PROGRAM MAIN
VAR CONSTANT
  Dofs : ARRAY [0..3] OF INT := [1, 3, 6, 7];
  IterationCount : INT := 5;
  TrajactoryCount : DINT := 64 * 1024;
END_VAR
VAR
  _positionDist : RandomGaussian(seed:=42, mu:=0, sigma:=4);
  _dynamicDist : RandomGaussian(seed:=43, mu:=0, sigma:=0.8);
  _limitDist : RandomUniform(seed:=44, lowerBound:=0, upperBound:=4);
  
  _p : Randomizer(_positionDist);
  _d : Randomizer(_dynamicDist);
  _l : Randomizer(_limitDist);
  
  _otg : Struckig.Ruckig(0.001);
  _input : Struckig.InputParameter(0);
  _output : Struckig.OutputParameter;
  
  _step : INT := 0;
  _dt, _it, _jt : DINT := 0;
  
  _trajectoryStatistic, _itStatistic, _worstStatistic : MovingStatistic;
  
  _averageMean, _worstMean, _averageSigma, _worstSigma : ARRAY[0..3] OF LREAL; 
  
  _cpucounter : Tc2_System.GETCPUACCOUNT;
END_VAR

REPEAT
  CASE _step
  OF
    // setup ****************************************************
    0: 
    // **********************************************************
      
      _input.FB_init(TRUE, TRUE, dofs:=Dofs[_dt]);
      _trajectoryStatistic.Reset();
      _itStatistic.Reset();
      _worstStatistic.Reset();
      
      _p.Fill(ADR(_input.CurrentPosition), Dofs[_dt]);
      _p.Fill(ADR(_input.TargetPosition), Dofs[_dt]);
      _l.FillMax(ADR(_input.maxVelocity), Dofs[_dt], ADR(_input.TargetVelocity));
      _l.FillMax(ADR(_input.maxAcceleration), Dofs[_dt], ADR(_input.TargetAcceleration));
      _l.Fill(ADR(_input.maxJerk), Dofs[_dt]);
      CheckCalculation(_otg, _input);  
    
      _step := 1;
  
    // iterate start ********************************************
    1: 
    // **********************************************************
    
      _trajectoryStatistic.Reset();
      _step := 2;
      
    // iterate loop *********************************************
    2: 
    // **********************************************************
    
      _p.Fill(ADR(_input.CurrentPosition), Dofs[_dt]);
      _d.FillOrZero(ADR(_input.CurrentVelocity), Dofs[_dt], 0.9);
      _d.FillOrZero(ADR(_input.CurrentAcceleration), Dofs[_dt], 0.8);
      _p.Fill(ADR(_input.TargetPosition), Dofs[_dt]);
      _d.FillOrZero(ADR(_input.TargetVelocity), Dofs[_dt], 0.7);
      _d.FillOrZero(ADR(_input.TargetAcceleration), Dofs[_dt], 0.6);
      _l.FillMax(ADR(_input.MaxVelocity), Dofs[_dt], ADR(_input.TargetVelocity));
      _l.FillMax(ADR(_input.MaxAcceleration), Dofs[_dt], ADR(_input.TargetAcceleration));
      _l.Fill(ADR(_input.MaxJerk), Dofs[_dt]);
  
      IF NOT _otg.ValidateInput(_input)
      THEN
        RETURN;
      END_IF
  
      _trajectoryStatistic.Append(CheckCalculation(_otg, _input));
      _jt := _jt + 1;
      IF _jt > TrajactoryCount
      THEN
        _it := _it + 1;
        _jt := 0;        
        _step := 1;
        _itStatistic.Append(_trajectoryStatistic.Mean);
        _worstStatistic.Append(_trajectoryStatistic.Maximum);
      END_IF
      
      IF _it > IterationCount
      THEN
        _step := 3;
      END_IF
      
    // iterate end **********************************************
    3: 
    // **********************************************************
    
      _it := 0;
      _jt := 0;
      _averageMean[_dt] := _itStatistic.Mean;
      _averageSigma[_dt] := _itStatistic.Sigma;
      _worstMean[_dt] := _worstStatistic.Mean;
      _worstSigma[_dt] := _worstStatistic.Sigma;      
      _dt := _dt + 1;
      _step := SEL(_dt > 3, 0, 4);

    // done******* **********************************************
    4: 
    // **********************************************************
      ; 
  END_CASE
UNTIL _step = 4 
AND_THEN TRUE // wtf, fix this already Beckhoff - no breakpoints without an additional condition!!!! 
END_REPEAT

_step := 4;

METHOD CheckCalculation : LREAL;
VAR_INPUT
  otg : REFERENCE TO Struckig.Ruckig;
  input : REFERENCE TO Struckig.InputParameter;
END_VAR
VAR
  output : Struckig.OutputParameter;
END_VAR
otg.update(input, output);
CheckCalculation := output.CalculationDuration;
END_METHOD

END_PROGRAM

(* stored: Version 1.1.0.1, ProductVersion 3.1.4024.9
   POU MAIN: Id {c24cf36f-30d9-4bef-a3e5-6c8b5a1b2c55}, SpecialFunc None
   Method CheckCalculation: Id {829178d5-91bc-4df1-995d-bbe41aca5758} *)
